FUNCTION_BLOCK HandlingSkill (* Basic FB with empty ECC *)
  (* Standard: 61499-2 *)
  (* Version 1.0, 2021-09-15, dorofeev *)
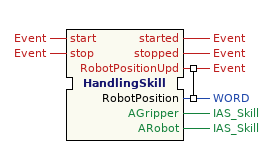
  EVENT_INPUT
    start;
    stop;
  END_EVENT
  EVENT_OUTPUT
    started;
    stopped;
    RobotPositionUpd WITH RobotPosition;
  END_EVENT
  VAR_OUTPUT
    RobotPosition : WORD;
  END_VAR
  PLUGS
    AGripper : IAS_Skill;
    ARobot : IAS_Skill;
  END_PLUGS
  EC_STATES
    START; (* Initial State *)
    State_1 : RobotGoTo1 -> RobotPositionUpd, -> ARobot.start, -> started;
    State_2 : -> AGripper.start;
    State_3 : RobotGoTo11 -> RobotPositionUpd, -> ARobot.start;
    State_4 : -> AGripper.start;
    State_5 : -> AGripper.start;
    State_6 : RobotGoTo12 -> RobotPositionUpd, -> ARobot.start;
    State_7 : RobotGoTo3 -> RobotPositionUpd, -> ARobot.start;
    State_8 : -> AGripper.start;
    State_9 : RobotGoTo13 -> RobotPositionUpd, -> ARobot.start;
    State_10 : RobotGoTo4 -> RobotPositionUpd, -> ARobot.start;
    State_11 : -> AGripper.start;
    State_12 : RobotGoTo14 -> RobotPositionUpd, -> ARobot.start;
    State_13 : RobotGoTo99 -> RobotPositionUpd, -> ARobot.start;
    State;
    State_15 : RobotGoTo2 -> RobotPositionUpd, -> ARobot.start;
    State_16 : -> AGripper.start;
    State_17;
    State_18;
    State_14;
    State_19;
    State_20;
    State_21;
    State_22;
    State_23;
    State_24;
    State_25;
    State_26;
    State_27;
    State_28 : -> AGripper.start;
    State_29;
    State_30;
    State_31;
    State_32 : -> AGripper.start;
    State_33;
    State_34 : -> stopped;
  END_STATES
  EC_TRANSITIONS
    State_13 TO State := ARobot.RSP[ARobot.currentState = "Executing"];
    State_9 TO State_17 := ARobot.RSP[ARobot.currentState = "Executing"];
    State_12 TO State_18 := ARobot.RSP[ARobot.currentState = "Executing"];
    START TO State_1 := start;
    State_1 TO State_14 := ARobot.RSP[ARobot.currentState = "Executing"];
    State_14 TO State_2 := ARobot.RSP[ARobot.currentState = "Idle"];
    State_2 TO State_19 := AGripper.RSP[AGripper.currentState = "Executing"];
    State_19 TO State_3 := AGripper.RSP[AGripper.currentState = "Idle"];
    State_3 TO State_20 := ARobot.RSP[ARobot.currentState = "Executing"];
    State_20 TO State_4 := ARobot.RSP[ARobot.currentState = "Idle"];
    State_4 TO State_21 := AGripper.RSP[AGripper.currentState = "Executing"];
    State_21 TO State_15 := AGripper.RSP[AGripper.currentState = "Idle"];
    State_15 TO State_22 := ARobot.RSP[ARobot.currentState = "Executing"];
    State_22 TO State_5 := ARobot.RSP[ARobot.currentState = "Idle"];
    State_5 TO State_23 := AGripper.RSP[AGripper.currentState = "Executing"];
    State_23 TO State_6 := AGripper.RSP[AGripper.currentState = "Idle"];
    State_6 TO State_24 := ARobot.RSP[ARobot.currentState = "Executing"];
    State_24 TO State_16 := ARobot.RSP[ARobot.currentState = "Idle"];
    State_16 TO State_25 := AGripper.RSP[AGripper.currentState = "Executing"];
    State_25 TO State_7 := AGripper.RSP[AGripper.currentState = "Idle"];
    State_7 TO State_26 := ARobot.RSP[ARobot.currentState = "Executing"];
    State_26 TO State_8 := ARobot.RSP[ARobot.currentState = "Idle"];
    State_8 TO State_27 := AGripper.RSP[AGripper.currentState = "Executing"];
    State_27 TO State_9 := AGripper.RSP[AGripper.currentState = "Idle"];
    State_17 TO State_28 := ARobot.RSP[ARobot.currentState = "Idle"];
    State_28 TO State_29 := AGripper.RSP[AGripper.currentState = "Executing"];
    State_29 TO State_10 := AGripper.RSP[AGripper.currentState = "Idle"];
    State_10 TO State_30 := ARobot.RSP[ARobot.currentState = "Executing"];
    State_30 TO State_11 := ARobot.RSP[ARobot.currentState = "Idle"];
    State_11 TO State_31 := AGripper.RSP[AGripper.currentState = "Executing"];
    State_31 TO State_12 := AGripper.RSP[AGripper.currentState = "Idle"];
    State_18 TO State_32 := ARobot.RSP[ARobot.currentState = "Idle"];
    State_32 TO State_33 := AGripper.RSP[AGripper.currentState = "Executing"];
    State_33 TO State_13 := AGripper.RSP[AGripper.currentState = "Idle"];
    State TO State_34 := ARobot.RSP[ARobot.currentState = "Idle"];
    State_34 TO START := 1;
  END_TRANSITIONS
  ALGORITHM RobotGoTo1 IN ST: (* New Algorithm *)
RobotPosition := 1;
  END_ALGORITHM
  ALGORITHM RobotGoTo2 IN ST: (* New Algorithm *)
RobotPosition := 2;
  END_ALGORITHM
  ALGORITHM RobotGoTo3 IN ST: (* New Algorithm *)
RobotPosition := 3;
  END_ALGORITHM
  ALGORITHM RobotGoTo4 IN ST: (* New Algorithm *)
RobotPosition := 4;
  END_ALGORITHM
  ALGORITHM RobotGoTo11 IN ST: (* New Algorithm *)
RobotPosition := 11;
  END_ALGORITHM
  ALGORITHM RobotGoTo12 IN ST: (* New Algorithm *)
RobotPosition := 12;
  END_ALGORITHM
  ALGORITHM RobotGoTo13 IN ST: (* New Algorithm *)
RobotPosition := 13;
  END_ALGORITHM
  ALGORITHM RobotGoTo14 IN ST: (* New Algorithm *)
RobotPosition := 14;
  END_ALGORITHM
  ALGORITHM RobotGoTo99 IN ST: (* New Algorithm *)
RobotPosition := 99;
  END_ALGORITHM
END_FUNCTION_BLOCK
